# EPICS IOC start-up script: iocsh/ethercatmcEL6688-PTP.iocsh
ethercatmcCreateAsynParam $(MOTOR_PORT) PTPState Int32
ethercatmcCreateAsynParam $(MOTOR_PORT) PTPOffset Int32
ethercatmcCreateAsynParam $(MOTOR_PORT) PTPSyncSeqNum Int32
ethercatmcCreateAsynParam $(MOTOR_PORT) SystemUTCtime Int64
ethercatmcCreateAsynParam $(MOTOR_PORT) DCTIME        Int64

dbLoadRecords("ethercatmcEL6688-PTP.template", "PREFIX=$(PREFIX), MOTOR_PORT=$(MOTOR_PORT)")
